// TIA Portal V20 export
TYPE "IO_AI"
   STRUCT
      IN : Struct
         ValueIn : Real;
      END_STRUCT;
   END_STRUCT;
END_TYPE
